ABB RAPID module: Module1.mod

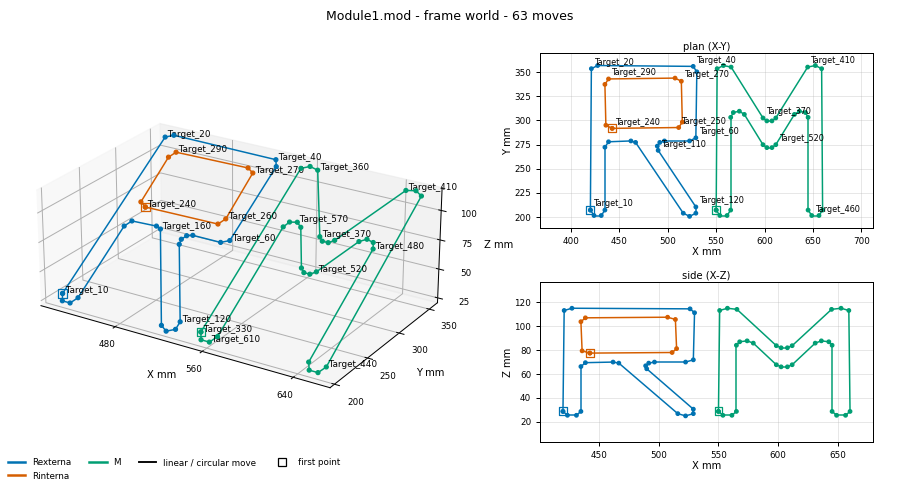
[picture p0: tool path of Module1.mod in frame world, 63 of 66 moves have a stored position in this frame; points joined in program order, loops and branches not executed]
MODULE Module1
        CONST robtarget Target_10:=[[20,222.5,-0.000045108],[0.707106781,-0.000000072,-0.000000072,-0.707106781],[0,0,0,0],[9E+09,9E+09,9E+09,9E+09,9E+09,9E+09]];
    CONST robtarget Target_20:=[[21.004809472,53.75,-0.000010897],[0.707106781,-0.000000072,-0.000000072,-0.707106781],[0,0,0,0],[9E+09,9E+09,9E+09,9E+09,9E+09,9E+09]];
    CONST robtarget Target_30:=[[27.5,50,-0.000010136],[0.707106781,-0.000000072,-0.000000072,-0.707106781],[0,0,0,0],[9E+09,9E+09,9E+09,9E+09,9E+09,9E+09]];
    CONST robtarget Target_40:=[[126.25,51.004809472,-0.00001034],[0.707106781,-0.000000072,-0.000000072,-0.707106781],[0,0,0,0],[9E+09,9E+09,9E+09,9E+09,9E+09,9E+09]];
    CONST robtarget Target_50:=[[130,57.5,-0.000011657],[0.707106781,-0.000000072,-0.000000072,-0.707106781],[0,0,0,0],[9E+09,9E+09,9E+09,9E+09,9E+09,9E+09]];
    CONST robtarget Target_60:=[[128.995190528,136.25,-0.000027622],[0.707106781,-0.000000072,-0.000000072,-0.707106781],[0,0,0,0],[9E+09,9E+09,9E+09,9E+09,9E+09,9E+09]];
    CONST robtarget Target_70:=[[122.5,140,-0.000028383],[0.707106781,-0.000000072,-0.000000072,-0.707106781],[0,0,0,0],[9E+09,9E+09,9E+09,9E+09,9E+09,9E+09]];
    CONST robtarget Target_80:=[[96.519237886,140,-0.000028383],[0.707106781,-0.000000072,-0.000000072,-0.707106781],[0,0,0,0],[9E+09,9E+09,9E+09,9E+09,9E+09,9E+09]];
    CONST robtarget Target_90:=[[91.698330814,141.754666677,-0.000028738],[0.707106781,-0.000000072,-0.000000072,-0.707106781],[0,0,0,0],[9E+09,9E+09,9E+09,9E+09,9E+09,9E+09]];
    CONST robtarget Target_100:=[[89.133179739,146.197638667,-0.000029638],[0.707106781,-0.000000072,-0.000000072,-0.707106781],[0,0,0,0],[9E+09,9E+09,9E+09,9E+09,9E+09,9E+09]];
    CONST robtarget Target_110:=[[90.024047358,151.25,-0.000030663],[0.707106781,-0.000000072,-0.000000072,-0.707106781],[0,0,0,0],[9E+09,9E+09,9E+09,9E+09,9E+09,9E+09]];
    CONST robtarget Target_120:=[[128.995190528,218.75,-0.000044348],[0.707106781,-0.000000072,-0.000000072,-0.707106781],[0,0,0,0],[9E+09,9E+09,9E+09,9E+09,9E+09,9E+09]];
    CONST robtarget Target_130:=[[128.995190528,226.25,-0.000045868],[0.707106781,-0.000000072,-0.000000072,-0.707106781],[0,0,0,0],[9E+09,9E+09,9E+09,9E+09,9E+09,9E+09]];
    CONST robtarget Target_140:=[[122.5,230,-0.000046628],[0.707106781,-0.000000072,-0.000000072,-0.707106781],[0,0,0,0],[9E+09,9E+09,9E+09,9E+09,9E+09,9E+09]];
    CONST robtarget Target_150:=[[116.004809472,226.25,-0.000045868],[0.707106781,-0.000000072,-0.000000072,-0.707106781],[0,0,0,0],[9E+09,9E+09,9E+09,9E+09,9E+09,9E+09]];
    CONST robtarget Target_160:=[[66.699128808,141.754666677,-0.000028738],[0.707106781,-0.000000072,-0.000000072,-0.707106781],[0,0,0,0],[9E+09,9E+09,9E+09,9E+09,9E+09,9E+09]];
    CONST robtarget Target_170:=[[61.878221735,140,-0.000028383],[0.707106781,-0.000000072,-0.000000072,-0.707106781],[0,0,0,0],[9E+09,9E+09,9E+09,9E+09,9E+09,9E+09]];
    CONST robtarget Target_180:=[[38.75,141.004809472,-0.000028586],[0.707106781,-0.000000072,-0.000000072,-0.707106781],[0,0,0,0],[9E+09,9E+09,9E+09,9E+09,9E+09,9E+09]];
    CONST robtarget Target_190:=[[35,147.5,-0.000029903],[0.707106781,-0.000000072,-0.000000072,-0.707106781],[0,0,0,0],[9E+09,9E+09,9E+09,9E+09,9E+09,9E+09]];
    CONST robtarget Target_200:=[[35,222.5,-0.000045108],[0.707106781,-0.000000072,-0.000000072,-0.707106781],[0,0,0,0],[9E+09,9E+09,9E+09,9E+09,9E+09,9E+09]];
    CONST robtarget Target_210:=[[31.25,228.995190528,-0.000046425],[0.707106781,-0.000000072,-0.000000072,-0.707106781],[0,0,0,0],[9E+09,9E+09,9E+09,9E+09,9E+09,9E+09]];
    CONST robtarget Target_220:=[[23.75,228.995190528,-0.000046425],[0.707106781,-0.000000072,-0.000000072,-0.707106781],[0,0,0,0],[9E+09,9E+09,9E+09,9E+09,9E+09,9E+09]];
    CONST robtarget Target_230:=[[20,222.5,-0.000045108],[0.707106781,-0.000000072,-0.000000072,-0.707106781],[0,0,0,0],[9E+09,9E+09,9E+09,9E+09,9E+09,9E+09]];
    CONST robtarget Target_240:=[[42.5,125,-0.000025341],[0.707106781,-0.000000072,-0.000000072,-0.707106781],[0,0,0,0],[9E+09,9E+09,9E+09,9E+09,9E+09,9E+09]];
    CONST robtarget Target_250:=[[111.25,123.995190529,-0.000025138],[0.707106781,-0.000000072,-0.000000072,-0.707106781],[0,0,0,0],[9E+09,9E+09,9E+09,9E+09,9E+09,9E+09]];
    CONST robtarget Target_260:=[[115,117.5,-0.000023821],[0.707106781,-0.000000072,-0.000000072,-0.707106781],[0,0,0,0],[9E+09,9E+09,9E+09,9E+09,9E+09,9E+09]];
    CONST robtarget Target_270:=[[113.995190528,68.75,-0.000013938],[0.707106781,-0.000000072,-0.000000072,-0.707106781],[0,0,0,0],[9E+09,9E+09,9E+09,9E+09,9E+09,9E+09]];
    CONST robtarget Target_280:=[[107.5,65,-0.000013178],[0.707106781,-0.000000072,-0.000000072,-0.707106781],[0,0,0,0],[9E+09,9E+09,9E+09,9E+09,9E+09,9E+09]];
    CONST robtarget Target_290:=[[38.75,66.004809471,-0.000013381],[0.707106781,-0.000000072,-0.000000072,-0.707106781],[0,0,0,0],[9E+09,9E+09,9E+09,9E+09,9E+09,9E+09]];
    CONST robtarget Target_300:=[[35,72.5,-0.000014698],[0.707106781,-0.000000072,-0.000000072,-0.707106781],[0,0,0,0],[9E+09,9E+09,9E+09,9E+09,9E+09,9E+09]];
    CONST robtarget Target_310:=[[36.004809472,121.25,-0.000024581],[0.707106781,-0.000000072,-0.000000072,-0.707106781],[0,0,0,0],[9E+09,9E+09,9E+09,9E+09,9E+09,9E+09]];
    CONST robtarget Target_320:=[[42.5,125,-0.000025341],[0.707106781,-0.000000072,-0.000000072,-0.707106781],[0,0,0,0],[9E+09,9E+09,9E+09,9E+09,9E+09,9E+09]];
    CONST robtarget Target_330:=[[150,222.5,-0.000045108],[0.707106781,-0.000000072,-0.000000072,-0.707106781],[0,0,0,0],[9E+09,9E+09,9E+09,9E+09,9E+09,9E+09]];
    CONST robtarget Target_340:=[[151.004809472,53.75,-0.000010897],[0.707106781,-0.000000072,-0.000000072,-0.707106781],[0,0,0,0],[9E+09,9E+09,9E+09,9E+09,9E+09,9E+09]];
    CONST robtarget Target_350:=[[157.5,50,-0.000010136],[0.707106781,-0.000000072,-0.000000072,-0.707106781],[0,0,0,0],[9E+09,9E+09,9E+09,9E+09,9E+09,9E+09]];
    CONST robtarget Target_360:=[[165.448538093,51.864224034,-0.000010515],[0.707106781,-0.000000072,-0.000000072,-0.707106781],[0,0,0,0],[9E+09,9E+09,9E+09,9E+09,9E+09,9E+09]];
    CONST robtarget Target_370:=[[198.382352941,112.591911765,-0.000022826],[0.707106781,-0.000000072,-0.000000072,-0.707106781],[0,0,0,0],[9E+09,9E+09,9E+09,9E+09,9E+09,9E+09]];
    CONST robtarget Target_380:=[[202.355980309,116.080987008,-0.000023533],[0.707106781,-0.000000072,-0.000000072,-0.707106781],[0,0,0,0],[9E+09,9E+09,9E+09,9E+09,9E+09,9E+09]];
    CONST robtarget Target_390:=[[207.644019691,116.080987008,-0.000023533],[0.707106781,-0.000000072,-0.000000072,-0.707106781],[0,0,0,0],[9E+09,9E+09,9E+09,9E+09,9E+09,9E+09]];
    CONST robtarget Target_400:=[[211.617647059,112.591911765,-0.000022826],[0.707106781,-0.000000072,-0.000000072,-0.707106781],[0,0,0,0],[9E+09,9E+09,9E+09,9E+09,9E+09,9E+09]];
    CONST robtarget Target_410:=[[244.551461907,51.864224034,-0.000010515],[0.707106781,-0.000000072,-0.000000072,-0.707106781],[0,0,0,0],[9E+09,9E+09,9E+09,9E+09,9E+09,9E+09]];
    CONST robtarget Target_420:=[[252.5,50,-0.000010136],[0.707106781,-0.000000072,-0.000000072,-0.707106781],[0,0,0,0],[9E+09,9E+09,9E+09,9E+09,9E+09,9E+09]];
    CONST robtarget Target_430:=[[258.995190528,53.75,-0.000010897],[0.707106781,-0.000000072,-0.000000072,-0.707106781],[0,0,0,0],[9E+09,9E+09,9E+09,9E+09,9E+09,9E+09]];
    CONST robtarget Target_440:=[[260,222.5,-0.000045108],[0.707106781,-0.000000072,-0.000000072,-0.707106781],[0,0,0,0],[9E+09,9E+09,9E+09,9E+09,9E+09,9E+09]];
    CONST robtarget Target_450:=[[256.25,228.995190528,-0.000046425],[0.707106781,-0.000000072,-0.000000072,-0.707106781],[0,0,0,0],[9E+09,9E+09,9E+09,9E+09,9E+09,9E+09]];
    CONST robtarget Target_460:=[[248.75,228.995190528,-0.000046425],[0.707106781,-0.000000072,-0.000000072,-0.707106781],[0,0,0,0],[9E+09,9E+09,9E+09,9E+09,9E+09,9E+09]];
    CONST robtarget Target_470:=[[245,222.5,-0.000045108],[0.707106781,-0.000000072,-0.000000072,-0.707106781],[0,0,0,0],[9E+09,9E+09,9E+09,9E+09,9E+09,9E+09]];
    CONST robtarget Target_480:=[[245,111.875,-0.00002268],[0.707106781,-0.000000072,-0.000000072,-0.707106781],[0,0,0,0],[9E+09,9E+09,9E+09,9E+09,9E+09,9E+09]];
    CONST robtarget Target_490:=[[242.256178199,106.075968276,-0.000021505],[0.707106781,-0.000000072,-0.000000072,-0.707106781],[0,0,0,0],[9E+09,9E+09,9E+09,9E+09,9E+09,9E+09]];
    CONST robtarget Target_500:=[[236.032328283,104.520005797,-0.00002119],[0.707106781,-0.000000072,-0.000000072,-0.707106781],[0,0,0,0],[9E+09,9E+09,9E+09,9E+09,9E+09,9E+09]];
    CONST robtarget Target_510:=[[230.882352941,108.345588236,-0.000021965],[0.707106781,-0.000000072,-0.000000072,-0.707106781],[0,0,0,0],[9E+09,9E+09,9E+09,9E+09,9E+09,9E+09]];
    CONST robtarget Target_520:=[[211.617647059,144.466911765,-0.000029289],[0.707106781,-0.000000072,-0.000000072,-0.707106781],[0,0,0,0],[9E+09,9E+09,9E+09,9E+09,9E+09,9E+09]];
    CONST robtarget Target_530:=[[207.644019691,147.955987007,-0.000029995],[0.707106781,-0.000000072,-0.000000072,-0.707106781],[0,0,0,0],[9E+09,9E+09,9E+09,9E+09,9E+09,9E+09]];
    CONST robtarget Target_540:=[[202.355980309,147.955987007,-0.000029995],[0.707106781,-0.000000072,-0.000000072,-0.707106781],[0,0,0,0],[9E+09,9E+09,9E+09,9E+09,9E+09,9E+09]];
    CONST robtarget Target_550:=[[198.382352941,144.466911765,-0.000029289],[0.707106781,-0.000000072,-0.000000072,-0.707106781],[0,0,0,0],[9E+09,9E+09,9E+09,9E+09,9E+09,9E+09]];
    CONST robtarget Target_560:=[[179.117647059,108.345588236,-0.000021965],[0.707106781,-0.000000072,-0.000000072,-0.707106781],[0,0,0,0],[9E+09,9E+09,9E+09,9E+09,9E+09,9E+09]];
    CONST robtarget Target_570:=[[173.967671717,104.520005797,-0.00002119],[0.707106781,-0.000000072,-0.000000072,-0.707106781],[0,0,0,0],[9E+09,9E+09,9E+09,9E+09,9E+09,9E+09]];
    CONST robtarget Target_580:=[[167.743821801,106.075968276,-0.000021505],[0.707106781,-0.000000072,-0.000000072,-0.707106781],[0,0,0,0],[9E+09,9E+09,9E+09,9E+09,9E+09,9E+09]];
    CONST robtarget Target_590:=[[165,111.875,-0.00002268],[0.707106781,-0.000000072,-0.000000072,-0.707106781],[0,0,0,0],[9E+09,9E+09,9E+09,9E+09,9E+09,9E+09]];
    CONST robtarget Target_600:=[[165,222.5,-0.000045108],[0.707106781,-0.000000072,-0.000000072,-0.707106781],[0,0,0,0],[9E+09,9E+09,9E+09,9E+09,9E+09,9E+09]];
    CONST robtarget Target_610:=[[161.25,228.995190528,-0.000046425],[0.707106781,-0.000000072,-0.000000072,-0.707106781],[0,0,0,0],[9E+09,9E+09,9E+09,9E+09,9E+09,9E+09]];
    CONST robtarget Target_620:=[[153.75,228.995190528,-0.000046425],[0.707106781,-0.000000072,-0.000000072,-0.707106781],[0,0,0,0],[9E+09,9E+09,9E+09,9E+09,9E+09,9E+09]];
    CONST robtarget Target_630:=[[150,222.5,-0.000045108],[0.707106781,-0.000000072,-0.000000072,-0.707106781],[0,0,0,0],[9E+09,9E+09,9E+09,9E+09,9E+09,9E+09]];
    CONST jointtarget Home:=[[0,0,0,0,0,0],[9E+09,9E+09,9E+09,9E+09,9E+09,9E+09]];
    CONST jointtarget Intermedio:=[[0,30,0,0,30,0],[9E+09,9E+09,9E+09,9E+09,9E+09,9E+09]];
    CONST jointtarget Mantenimiento:=[[74,42,-68,-4,12,0],[9E+09,9E+09,9E+09,9E+09,9E+09,9E+09]];
!***********************************************************
    !
    ! Módulo:  Module1
    !
    ! Descripción:
    !   <Introduzca la descripción aquí>
    !
    ! Autor: rinco
    !
    ! Versión: 1.0
    !
    !***********************************************************


    !***********************************************************
    !
    ! Procedimiento Main
    !
    !   Este es el punto de entrada de su programa
    !
    !***********************************************************
    PROC main()
        !Añada aquí su código
        WaitDI DI10_1, 1;
        IrAHome;
        IrAIntermedio;
        Rexterna;
        IrAIntermedio;
        Rinterna;
        IrAIntermedio;
        M;
        IrAIntermedio;
        IrAHome;
        SetDO DO10_1, 1;

        WaitDI DI10_2, 1;
        IrAHome;
        IrAMantenimiento;
        SetDO DO10_1, 0;




    ENDPROC
    PROC Rexterna()
        MoveL Target_10,v100,z10,HmarcadorFinal\WObj:=Tablero;
        MoveL Target_20,v100,z10,HmarcadorFinal\WObj:=Tablero;
        MoveL Target_30,v100,z10,HmarcadorFinal\WObj:=Tablero;
        MoveL Target_40,v100,z10,HmarcadorFinal\WObj:=Tablero;
        MoveL Target_50,v100,z10,HmarcadorFinal\WObj:=Tablero;
        MoveL Target_60,v100,z10,HmarcadorFinal\WObj:=Tablero;
        MoveL Target_70,v100,z10,HmarcadorFinal\WObj:=Tablero;
        MoveL Target_80,v100,z10,HmarcadorFinal\WObj:=Tablero;
        MoveL Target_90,v100,z10,HmarcadorFinal\WObj:=Tablero;
        MoveL Target_100,v100,z10,HmarcadorFinal\WObj:=Tablero;
        MoveL Target_110,v100,z10,HmarcadorFinal\WObj:=Tablero;
        MoveL Target_120,v100,z10,HmarcadorFinal\WObj:=Tablero;
        MoveL Target_130,v100,z10,HmarcadorFinal\WObj:=Tablero;
        MoveL Target_140,v100,z10,HmarcadorFinal\WObj:=Tablero;
        MoveL Target_150,v100,z10,HmarcadorFinal\WObj:=Tablero;
        MoveL Target_160,v100,z10,HmarcadorFinal\WObj:=Tablero;
        MoveL Target_170,v100,z10,HmarcadorFinal\WObj:=Tablero;
        MoveL Target_180,v100,z10,HmarcadorFinal\WObj:=Tablero;
        MoveL Target_190,v100,z10,HmarcadorFinal\WObj:=Tablero;
        MoveL Target_200,v100,z10,HmarcadorFinal\WObj:=Tablero;
        MoveL Target_210,v100,z10,HmarcadorFinal\WObj:=Tablero;
        MoveL Target_220,v100,z10,HmarcadorFinal\WObj:=Tablero;
        MoveL Target_230,v100,z10,HmarcadorFinal\WObj:=Tablero;
    ENDPROC
    PROC Rinterna()
        MoveL Target_240,v100,z10,HmarcadorFinal\WObj:=Tablero;
        MoveL Target_250,v100,z10,HmarcadorFinal\WObj:=Tablero;
        MoveL Target_260,v100,z10,HmarcadorFinal\WObj:=Tablero;
        MoveL Target_270,v100,z10,HmarcadorFinal\WObj:=Tablero;
        MoveL Target_280,v100,z10,HmarcadorFinal\WObj:=Tablero;
        MoveL Target_290,v100,z10,HmarcadorFinal\WObj:=Tablero;
        MoveL Target_300,v100,z10,HmarcadorFinal\WObj:=Tablero;
        MoveL Target_310,v100,z10,HmarcadorFinal\WObj:=Tablero;
        MoveL Target_320,v100,z10,HmarcadorFinal\WObj:=Tablero;
    ENDPROC
    PROC M()
        MoveL Target_330,v100,z10,HmarcadorFinal\WObj:=Tablero;
        MoveL Target_340,v100,z10,HmarcadorFinal\WObj:=Tablero;
        MoveL Target_350,v100,z10,HmarcadorFinal\WObj:=Tablero;
        MoveL Target_360,v100,z10,HmarcadorFinal\WObj:=Tablero;
        MoveL Target_370,v100,z10,HmarcadorFinal\WObj:=Tablero;
        MoveL Target_380,v100,z10,HmarcadorFinal\WObj:=Tablero;
        MoveL Target_390,v100,z10,HmarcadorFinal\WObj:=Tablero;
        MoveL Target_400,v100,z10,HmarcadorFinal\WObj:=Tablero;
        MoveL Target_410,v100,z10,HmarcadorFinal\WObj:=Tablero;
        MoveL Target_420,v100,z10,HmarcadorFinal\WObj:=Tablero;
        MoveL Target_430,v100,z10,HmarcadorFinal\WObj:=Tablero;
        MoveL Target_440,v100,z10,HmarcadorFinal\WObj:=Tablero;
        MoveL Target_450,v100,z10,HmarcadorFinal\WObj:=Tablero;
        MoveL Target_460,v100,z10,HmarcadorFinal\WObj:=Tablero;
        MoveL Target_470,v100,z10,HmarcadorFinal\WObj:=Tablero;
        MoveL Target_480,v100,z10,HmarcadorFinal\WObj:=Tablero;
        MoveL Target_490,v100,z10,HmarcadorFinal\WObj:=Tablero;
        MoveL Target_500,v100,z10,HmarcadorFinal\WObj:=Tablero;
        MoveL Target_510,v100,z10,HmarcadorFinal\WObj:=Tablero;
        MoveL Target_520,v100,z10,HmarcadorFinal\WObj:=Tablero;
        MoveL Target_530,v100,z10,HmarcadorFinal\WObj:=Tablero;
        MoveL Target_540,v100,z10,HmarcadorFinal\WObj:=Tablero;
        MoveL Target_550,v100,z10,HmarcadorFinal\WObj:=Tablero;
        MoveL Target_560,v100,z10,HmarcadorFinal\WObj:=Tablero;
        MoveL Target_570,v100,z10,HmarcadorFinal\WObj:=Tablero;
        MoveL Target_580,v100,z10,HmarcadorFinal\WObj:=Tablero;
        MoveL Target_590,v100,z10,HmarcadorFinal\WObj:=Tablero;
        MoveL Target_600,v100,z10,HmarcadorFinal\WObj:=Tablero;
        MoveL Target_610,v100,z10,HmarcadorFinal\WObj:=Tablero;
        MoveL Target_620,v100,z10,HmarcadorFinal\WObj:=Tablero;
        MoveL Target_630,v100,z10,HmarcadorFinal\WObj:=Tablero;
    ENDPROC
    PROC IrAHome()
        MoveAbsJ Home,v100,z100,HmarcadorFinal\WObj:=Tablero;
    ENDPROC
    PROC IrAIntermedio()
        MoveAbsJ Intermedio,v100,z100,HmarcadorFinal\WObj:=Tablero;
    ENDPROC
    PROC IrAMantenimiento()
        MoveAbsJ Mantenimiento,v100,z100,HmarcadorFinal\WObj:=Tablero;
    ENDPROC
ENDMODULE
